PROGRAM P_System
VAR
	_arrFbButton:			ARRAY[0..10] OF FB_Button;
	_arrTon:				ARRAY[0..10] OF TON;
	_fbCT:					FB_CycleTime1;
	_cttime:				REAL;
	
	_rTRIG:					R_TRIG;
	_iProductionCount:      INT;//产能计数
	_bCountZero:			BOOL;//产能计数清零
END_VAR

A_Machine();
A_System();

ACTION A_Machine:
//CT测试
_fbCT(Execute:=G_arrCylinder[E_Cylinder.TakeUcLift].stOutput.bWork, CycleTime=> );
_cttime:=TIME_TO_REAL(_fbCT.CycleTime)/1000;
//复位 退出空跑模式
IF G_stSystem.stInput.bReset THEN
	GVL.stSetting.bDryRun:=FALSE;
END_IF

//产能计数
_rTRIG(CLK:= G_arrCylinder[E_Cylinder.OpenLockLift].stOutput.bWork, Q=> );
IF G_stSystem.stMode.bAutoRunning AND NOT GVL.stSetting.bDryRun AND _rTRIG.Q THEN
	_iProductionCount:=_iProductionCount+1;
END_IF
IF NOT G_stSystem.stMode.bAutoRunning  AND  _bCountZero THEN
	_iProductionCount:=0;
END_IF
END_ACTION

ACTION A_System:
G_stSystem.stInput.bEStop:=NOT GVL.I.bEStop;
_arrTon[0](IN:=GVL.I.bResetAlarm,PT:=T#3S , Q=>G_stSystem.stInput.bInit , ET=> );


GVL.Q.bBeacon_Buzzer:=G_stSystem.stOutput.bLightRed AND NOT MachineManage.G_stSystem.stInput.bQuiet;
GVL.Q.bRuning:=GVL.Q.bBeacon_Green:=G_stSystem.stOutput.bLightGreen;
GVL.Q.bStop:=GVL.Q.bBeacon_Red:=G_stSystem.stOutput.bLightRed;
GVL.Q.bBeacon_Yellow:=G_stSystem.stOutput.bLightYellow;

_arrFbButton[0](In:=G_stSystem.stInput.bStart, CLK:=GVL.I.bStart );
_arrFbButton[1](In:= G_stSystem.stInput.bStop, CLK:=GVL.I.bStop );
_arrFbButton[2](In:=G_stSystem.stInput.bResetAlarm , CLK:= GVL.I.bResetAlarm  );

G_stSystem.stLogConfig.bExecute:=TRUE;
G_stSystem.stLogConfig.sFilePath:='D:\PLC\Log\System';

P_Machine(StationCount:=E_Station.Length);
END_ACTION

END_PROGRAM

(* stored: Version 1.1.0.1, ProductVersion 3.1.4024.3
   POU P_System: Id {ad3eb28e-c698-41e7-a998-ab791339b3bf}, SpecialFunc None
   Action A_Machine: Id {bad766d9-b53e-4b69-8971-767e1991fe7c}
   Action A_System: Id {ac834835-5c48-436c-baed-30b007fe8f96} *)
